Yaskawa INFORM job: LT.JBI

/JOB
//NAME LT
//POS
///NPOS 0,0,0,0,0,0
//INST
///DATE 2023/06/06 13:07
///ATTR SC,RW,MC
///GROUP1 RB1,BS1
///LVARS 5,2,0,0,0,1,1,0
NOP
'=== initialize ===
'--- LT mode ---------------
GETARG LB000 IARG#(1)
'--- LT func. file# --------
GETARG LB001 IARG#(2)
JUMP *OFF IF LB000=0
JUMP *ON IF LB000=1
JUMP *END
*ON
SKILLSND "LTRACKOF"
ADVINIT
SKILLSND "LTRACKON LT:1"
JUMP *END
*OFF
SKILLSND "LSRCHOF"
SKILLSND "LTRACKOF"
ADVINIT
JUMP *END
*END
END
